//     Term 9 (AT2000-0250)/CC Outputs/Current setpoint value Ch.5 <-> Data Pointer/CurrentSetpointValues[4]
//     Term 9 (AT2000-0250)/CC Outputs/Current setpoint value Ch.6 <-> Data Pointer/CurrentSetpointValues[5]
//     Term 9 (AT2000-0250)/CC Outputs/Current setpoint value Ch.7 <-> Data Pointer/CurrentSetpointValues[6]
//     Term 9 (AT2000-0250)/CC Outputs/Current setpoint value Ch.8 <-> Data Pointer/CurrentSetpointValues[7]
//     Term 9 (AT2000-0250)/CC Outputs/Current setpoint value Ch.9 <-> Data Pointer/CurrentSetpointValues[8]
//     Term 9 (AT2000-0250)/Term 10 (AT2000-5250)/FB Inputs/Value Channel 01 <-> Data Pointer/RawPositionValues[0]
//     Term 9 (AT2000-0250)/Term 10 (AT2000-5250)/FB Inputs/Value Channel 02 <-> Data Pointer/RawPositionValues[1]
//     Term 9 (AT2000-0250)/Term 10 (AT2000-5250)/FB Inputs/Value Channel 03 <-> Data Pointer/RawPositionValues[2]
//     Term 9 (AT2000-0250)/Term 10 (AT2000-5250)/FB Inputs/Value Channel 04 <-> Data Pointer/RawPositionValues[3]
//     Term 9 (AT2000-0250)/Term 10 (AT2000-5250)/FB Inputs/Value Channel 05 <-> Data Pointer/RawPositionValues[4]
//     Term 9 (AT2000-0250)/Term 10 (AT2000-5250)/FB Inputs/Value Channel 06 <-> Data Pointer/RawPositionValues[5]
//     Term 9 (AT2000-0250)/Term 10 (AT2000-5250)/FB Inputs/Value Channel 07 <-> Data Pointer/RawPositionValues[6]
//     Term 9 (AT2000-0250)/Term 10 (AT2000-5250)/FB Inputs/Value Channel 08 <-> Data Pointer/RawPositionValues[7]
//     Term 9 (AT2000-0250)/Term 10 (AT2000-5250)/FB Inputs/Value Channel 09 <-> Data Pointer/RawPositionValues[8]
//     Term 9 (AT2000-0250)/Term 10 (AT2000-5250)/FB Inputs/Value Channel 10 <-> Data Pointer/RawPositionValues[9]
//     Term 9 (AT2000-0250)/Term 10 (AT2000-5250)/FB Inputs/Value Channel 11 <-> Data Pointer/RawPositionValues[10]
//     Term 9 (AT2000-0250)/Term 10 (AT2000-5250)/FB Inputs/Value Channel 12 <-> Data Pointer/RawPositionValues[11]
//     Term 9 (AT2000-0250)/Term 10 (AT2000-5250)/FB Inputs/Value Channel 13 <-> Data Pointer/RawPositionValues[12]
//     Term 9 (AT2000-0250)/Term 10 (AT2000-5250)/FB Inputs/Value Channel 14 <-> Data Pointer/RawPositionValues[13]
//     Term 9 (AT2000-0250)/Term 10 (AT2000-5250)/FB Inputs/Value Channel 15 <-> Data Pointer/RawPositionValues[14]
//     Term 9 (AT2000-0250)/Term 10 (AT2000-5250)/FB Inputs/Value Channel 16 <-> Data Pointer/RawPositionValues[15]
//     Term 9 (AT2000-0250)/Term 10 (AT2000-5250)/FB Inputs/Value Channel 17 <-> Data Pointer/RawPositionValues[16]
//     Term 9 (AT2000-0250)/Term 10 (AT2000-5250)/FB Inputs/Value Channel 18 <-> Data Pointer/RawPositionValues[17]
//     Term 9 (AT2000-0250)/Term 10 (AT2000-5250)/FB Inputs/Value Channel 19 <-> Data Pointer/RawPositionValues[18]
//     Term 9 (AT2000-0250)/Term 10 (AT2000-5250)/FB Inputs/Value Channel 20 <-> Data Pointer/RawPositionValues[19]
//     Term 9 (AT2000-0250)/Term 10 (AT2000-5250)/FB Inputs/Value Channel 21 <-> Data Pointer/RawPositionValues[20]
//     Term 9 (AT2000-0250)/Term 10 (AT2000-5250)/FB Inputs/Value Channel 22 <-> Data Pointer/RawPositionValues[21]
//     Term 9 (AT2000-0250)/Term 10 (AT2000-5250)/FB Inputs/Value Channel 23 <-> Data Pointer/RawPositionValues[22]
//     Term 9 (AT2000-0250)/Term 10 (AT2000-5250)/FB Inputs/Value Channel 24 <-> Data Pointer/RawPositionValues[23]
//     Term 9 (AT2000-0250)/Term 10 (AT2000-5250)/FB Inputs/Value Channel 25 <-> Data Pointer/RawPositionValues[24]
//     Term 9 (AT2000-0250)/Term 10 (AT2000-5250)/FB Inputs/Value Channel 26 <-> Data Pointer/RawPositionValues[25]
//     Term 9 (AT2000-0250)/Term 10 (AT2000-5250)/FB Inputs/Value Channel 27 <-> Data Pointer/RawPositionValues[26]
//     Term 9 (AT2000-0250)/Term 10 (AT2000-5250)/FB Inputs/Value Channel 28 <-> Data Pointer/RawPositionValues[27]
//     Term 9 (AT2000-0250)/Term 10 (AT2000-5250)/FB Inputs/Value Channel 29 <-> Data Pointer/RawPositionValues[28]
//     Term 9 (AT2000-0250)/Term 10 (AT2000-5250)/FB Inputs/Value Channel 30 <-> Data Pointer/RawPositionValues[29]
//     Term 9 (AT2000-0250)/Term 10 (AT2000-5250)/FB Inputs/Value Channel 31 <-> Data Pointer/RawPositionValues[30]
//     Term 9 (AT2000-0250)/Term 10 (AT2000-5250)/FB Inputs/Value Channel 32 <-> Data Pointer/RawPositionValues[31]
//   (this object) <-> TcCOM Objects/XtsProcessingUnit 1/Part 1/Module 6
//     Term 11 (AT2000-0250)/CC Inputs/Current actual value Ch.1 <-> Data Pointer/CurrentActualValues[0]
//     Term 11 (AT2000-0250)/CC Inputs/Current actual value Ch.10 <-> Data Pointer/CurrentActualValues[9]
//     Term 11 (AT2000-0250)/CC Inputs/Current actual value Ch.11 <-> Data Pointer/CurrentActualValues[10]
//     Term 11 (AT2000-0250)/CC Inputs/Current actual value Ch.12 <-> Data Pointer/CurrentActualValues[11]
//     Term 11 (AT2000-0250)/CC Inputs/Current actual value Ch.13 <-> Data Pointer/CurrentActualValues[12]
//     Term 11 (AT2000-0250)/CC Inputs/Current actual value Ch.14 <-> Data Pointer/CurrentActualValues[13]
//     Term 11 (AT2000-0250)/CC Inputs/Current actual value Ch.15 <-> Data Pointer/CurrentActualValues[14]
//     Term 11 (AT2000-0250)/CC Inputs/Current actual value Ch.2 <-> Data Pointer/CurrentActualValues[1]
//     Term 11 (AT2000-0250)/CC Inputs/Current actual value Ch.3 <-> Data Pointer/CurrentActualValues[2]
//     Term 11 (AT2000-0250)/CC Inputs/Current actual value Ch.4 <-> Data Pointer/CurrentActualValues[3]
//     Term 11 (AT2000-0250)/CC Inputs/Current actual value Ch.5 <-> Data Pointer/CurrentActualValues[4]
//     Term 11 (AT2000-0250)/CC Inputs/Current actual value Ch.6 <-> Data Pointer/CurrentActualValues[5]
//     Term 11 (AT2000-0250)/CC Inputs/Current actual value Ch.7 <-> Data Pointer/CurrentActualValues[6]
//     Term 11 (AT2000-0250)/CC Inputs/Current actual value Ch.8 <-> Data Pointer/CurrentActualValues[7]
//     Term 11 (AT2000-0250)/CC Inputs/Current actual value Ch.9 <-> Data Pointer/CurrentActualValues[8]
//     Term 11 (AT2000-0250)/CC Inputs/Status <-> Data Pointer/Status
//     Term 11 (AT2000-0250)/CC Outputs/Control <-> Data Pointer/Control
//     Term 11 (AT2000-0250)/CC Outputs/Current setpoint value Ch.1 <-> Data Pointer/CurrentSetpointValues[0]
//     Term 11 (AT2000-0250)/CC Outputs/Current setpoint value Ch.10 <-> Data Pointer/CurrentSetpointValues[9]
//     Term 11 (AT2000-0250)/CC Outputs/Current setpoint value Ch.11 <-> Data Pointer/CurrentSetpointValues[10]
//     Term 11 (AT2000-0250)/CC Outputs/Current setpoint value Ch.12 <-> Data Pointer/CurrentSetpointValues[11]
//     Term 11 (AT2000-0250)/CC Outputs/Current setpoint value Ch.13 <-> Data Pointer/CurrentSetpointValues[12]
//     Term 11 (AT2000-0250)/CC Outputs/Current setpoint value Ch.14 <-> Data Pointer/CurrentSetpointValues[13]
//     Term 11 (AT2000-0250)/CC Outputs/Current setpoint value Ch.15 <-> Data Pointer/CurrentSetpointValues[14]
//     Term 11 (AT2000-0250)/CC Outputs/Current setpoint value Ch.2 <-> Data Pointer/CurrentSetpointValues[1]
//     Term 11 (AT2000-0250)/CC Outputs/Current setpoint value Ch.3 <-> Data Pointer/CurrentSetpointValues[2]
//     Term 11 (AT2000-0250)/CC Outputs/Current setpoint value Ch.4 <-> Data Pointer/CurrentSetpointValues[3]
//     Term 11 (AT2000-0250)/CC Outputs/Current setpoint value Ch.5 <-> Data Pointer/CurrentSetpointValues[4]
//     Term 11 (AT2000-0250)/CC Outputs/Current setpoint value Ch.6 <-> Data Pointer/CurrentSetpointValues[5]
//     Term 11 (AT2000-0250)/CC Outputs/Current setpoint value Ch.7 <-> Data Pointer/CurrentSetpointValues[6]
//     Term 11 (AT2000-0250)/CC Outputs/Current setpoint value Ch.8 <-> Data Pointer/CurrentSetpointValues[7]
//     Term 11 (AT2000-0250)/CC Outputs/Current setpoint value Ch.9 <-> Data Pointer/CurrentSetpointValues[8]
//     Term 11 (AT2000-0250)/Term 12 (AT2000-5250)/FB Inputs/Value Channel 01 <-> Data Pointer/RawPositionValues[0]
//     Term 11 (AT2000-0250)/Term 12 (AT2000-5250)/FB Inputs/Value Channel 02 <-> Data Pointer/RawPositionValues[1]
//     Term 11 (AT2000-0250)/Term 12 (AT2000-5250)/FB Inputs/Value Channel 03 <-> Data Pointer/RawPositionValues[2]
//     Term 11 (AT2000-0250)/Term 12 (AT2000-5250)/FB Inputs/Value Channel 04 <-> Data Pointer/RawPositionValues[3]
//     Term 11 (AT2000-0250)/Term 12 (AT2000-5250)/FB Inputs/Value Channel 05 <-> Data Pointer/RawPositionValues[4]
//     Term 11 (AT2000-0250)/Term 12 (AT2000-5250)/FB Inputs/Value Channel 06 <-> Data Pointer/RawPositionValues[5]
//     Term 11 (AT2000-0250)/Term 12 (AT2000-5250)/FB Inputs/Value Channel 07 <-> Data Pointer/RawPositionValues[6]
//     Term 11 (AT2000-0250)/Term 12 (AT2000-5250)/FB Inputs/Value Channel 08 <-> Data Pointer/RawPositionValues[7]
//     Term 11 (AT2000-0250)/Term 12 (AT2000-5250)/FB Inputs/Value Channel 09 <-> Data Pointer/RawPositionValues[8]
//     Term 11 (AT2000-0250)/Term 12 (AT2000-5250)/FB Inputs/Value Channel 10 <-> Data Pointer/RawPositionValues[9]
//     Term 11 (AT2000-0250)/Term 12 (AT2000-5250)/FB Inputs/Value Channel 11 <-> Data Pointer/RawPositionValues[10]
//     Term 11 (AT2000-0250)/Term 12 (AT2000-5250)/FB Inputs/Value Channel 12 <-> Data Pointer/RawPositionValues[11]
//     Term 11 (AT2000-0250)/Term 12 (AT2000-5250)/FB Inputs/Value Channel 13 <-> Data Pointer/RawPositionValues[12]
//     Term 11 (AT2000-0250)/Term 12 (AT2000-5250)/FB Inputs/Value Channel 14 <-> Data Pointer/RawPositionValues[13]
//     Term 11 (AT2000-0250)/Term 12 (AT2000-5250)/FB Inputs/Value Channel 15 <-> Data Pointer/RawPositionValues[14]
//     Term 11 (AT2000-0250)/Term 12 (AT2000-5250)/FB Inputs/Value Channel 16 <-> Data Pointer/RawPositionValues[15]
//     Term 11 (AT2000-0250)/Term 12 (AT2000-5250)/FB Inputs/Value Channel 17 <-> Data Pointer/RawPositionValues[16]
//     Term 11 (AT2000-0250)/Term 12 (AT2000-5250)/FB Inputs/Value Channel 18 <-> Data Pointer/RawPositionValues[17]
//     Term 11 (AT2000-0250)/Term 12 (AT2000-5250)/FB Inputs/Value Channel 19 <-> Data Pointer/RawPositionValues[18]
//     Term 11 (AT2000-0250)/Term 12 (AT2000-5250)/FB Inputs/Value Channel 20 <-> Data Pointer/RawPositionValues[19]
//     Term 11 (AT2000-0250)/Term 12 (AT2000-5250)/FB Inputs/Value Channel 21 <-> Data Pointer/RawPositionValues[20]
//     Term 11 (AT2000-0250)/Term 12 (AT2000-5250)/FB Inputs/Value Channel 22 <-> Data Pointer/RawPositionValues[21]
//     Term 11 (AT2000-0250)/Term 12 (AT2000-5250)/FB Inputs/Value Channel 23 <-> Data Pointer/RawPositionValues[22]
//     Term 11 (AT2000-0250)/Term 12 (AT2000-5250)/FB Inputs/Value Channel 24 <-> Data Pointer/RawPositionValues[23]
//     Term 11 (AT2000-0250)/Term 12 (AT2000-5250)/FB Inputs/Value Channel 25 <-> Data Pointer/RawPositionValues[24]
//     Term 11 (AT2000-0250)/Term 12 (AT2000-5250)/FB Inputs/Value Channel 26 <-> Data Pointer/RawPositionValues[25]
//     Term 11 (AT2000-0250)/Term 12 (AT2000-5250)/FB Inputs/Value Channel 27 <-> Data Pointer/RawPositionValues[26]
//     Term 11 (AT2000-0250)/Term 12 (AT2000-5250)/FB Inputs/Value Channel 28 <-> Data Pointer/RawPositionValues[27]
//     Term 11 (AT2000-0250)/Term 12 (AT2000-5250)/FB Inputs/Value Channel 29 <-> Data Pointer/RawPositionValues[28]
//     Term 11 (AT2000-0250)/Term 12 (AT2000-5250)/FB Inputs/Value Channel 30 <-> Data Pointer/RawPositionValues[29]
//     Term 11 (AT2000-0250)/Term 12 (AT2000-5250)/FB Inputs/Value Channel 31 <-> Data Pointer/RawPositionValues[30]
//     Term 11 (AT2000-0250)/Term 12 (AT2000-5250)/FB Inputs/Value Channel 32 <-> Data Pointer/RawPositionValues[31]
//   (this object) <-> TcCOM Objects/XtsProcessingUnit 1/Part 1/Module 7
//     Term 13 (AT2050-0500)/CC Inputs/Current actual value Ch.1 <-> Data Pointer/CurrentActualValues[0]
//     Term 13 (AT2050-0500)/CC Inputs/Current actual value Ch.10 <-> Data Pointer/CurrentActualValues[9]
//     Term 13 (AT2050-0500)/CC Inputs/Current actual value Ch.11 <-> Data Pointer/CurrentActualValues[10]
//     Term 13 (AT2050-0500)/CC Inputs/Current actual value Ch.12 <-> Data Pointer/CurrentActualValues[11]
//     Term 13 (AT2050-0500)/CC Inputs/Current actual value Ch.13 <-> Data Pointer/CurrentActualValues[12]
//     Term 13 (AT2050-0500)/CC Inputs/Current actual value Ch.14 <-> Data Pointer/CurrentActualValues[13]
//     Term 13 (AT2050-0500)/CC Inputs/Current actual value Ch.15 <-> Data Pointer/CurrentActualValues[14]
//     Term 13 (AT2050-0500)/CC Inputs/Current actual value Ch.2 <-> Data Pointer/CurrentActualValues[1]
//     Term 13 (AT2050-0500)/CC Inputs/Current actual value Ch.3 <-> Data Pointer/CurrentActualValues[2]
//     Term 13 (AT2050-0500)/CC Inputs/Current actual value Ch.4 <-> Data Pointer/CurrentActualValues[3]
//     Term 13 (AT2050-0500)/CC Inputs/Current actual value Ch.5 <-> Data Pointer/CurrentActualValues[4]
//     Term 13 (AT2050-0500)/CC Inputs/Current actual value Ch.6 <-> Data Pointer/CurrentActualValues[5]
//     Term 13 (AT2050-0500)/CC Inputs/Current actual value Ch.7 <-> Data Pointer/CurrentActualValues[6]
//     Term 13 (AT2050-0500)/CC Inputs/Current actual value Ch.8 <-> Data Pointer/CurrentActualValues[7]
//     Term 13 (AT2050-0500)/CC Inputs/Current actual value Ch.9 <-> Data Pointer/CurrentActualValues[8]
//     Term 13 (AT2050-0500)/CC Inputs/Status <-> Data Pointer/Status
//     Term 13 (AT2050-0500)/CC Outputs/Control <-> Data Pointer/Control
//     Term 13 (AT2050-0500)/CC Outputs/Current setpoint value Ch.1 <-> Data Pointer/CurrentSetpointValues[0]
//     Term 13 (AT2050-0500)/CC Outputs/Current setpoint value Ch.10 <-> Data Pointer/CurrentSetpointValues[9]
//     Term 13 (AT2050-0500)/CC Outputs/Current setpoint value Ch.11 <-> Data Pointer/CurrentSetpointValues[10]
//     Term 13 (AT2050-0500)/CC Outputs/Current setpoint value Ch.12 <-> Data Pointer/CurrentSetpointValues[11]
//     Term 13 (AT2050-0500)/CC Outputs/Current setpoint value Ch.13 <-> Data Pointer/CurrentSetpointValues[12]
//     Term 13 (AT2050-0500)/CC Outputs/Current setpoint value Ch.14 <-> Data Pointer/CurrentSetpointValues[13]
//     Term 13 (AT2050-0500)/CC Outputs/Current setpoint value Ch.15 <-> Data Pointer/CurrentSetpointValues[14]
//     Term 13 (AT2050-0500)/CC Outputs/Current setpoint value Ch.2 <-> Data Pointer/CurrentSetpointValues[1]
//     Term 13 (AT2050-0500)/CC Outputs/Current setpoint value Ch.3 <-> Data Pointer/CurrentSetpointValues[2]
//     Term 13 (AT2050-0500)/CC Outputs/Current setpoint value Ch.4 <-> Data Pointer/CurrentSetpointValues[3]
//     Term 13 (AT2050-0500)/CC Outputs/Current setpoint value Ch.5 <-> Data Pointer/CurrentSetpointValues[4]
//     Term 13 (AT2050-0500)/CC Outputs/Current setpoint value Ch.6 <-> Data Pointer/CurrentSetpointValues[5]
//     Term 13 (AT2050-0500)/CC Outputs/Current setpoint value Ch.7 <-> Data Pointer/CurrentSetpointValues[6]
//     Term 13 (AT2050-0500)/CC Outputs/Current setpoint value Ch.8 <-> Data Pointer/CurrentSetpointValues[7]
//     Term 13 (AT2050-0500)/CC Outputs/Current setpoint value Ch.9 <-> Data Pointer/CurrentSetpointValues[8]
//     Term 13 (AT2050-0500)/Term 14 (AT2050-5500)/FB Inputs/Value Channel 01 <-> Data Pointer/RawPositionValues[0]
//     Term 13 (AT2050-0500)/Term 14 (AT2050-5500)/FB Inputs/Value Channel 02 <-> Data Pointer/RawPositionValues[1]
//     Term 13 (AT2050-0500)/Term 14 (AT2050-5500)/FB Inputs/Value Channel 03 <-> Data Pointer/RawPositionValues[2]
//     Term 13 (AT2050-0500)/Term 14 (AT2050-5500)/FB Inputs/Value Channel 04 <-> Data Pointer/RawPositionValues[3]
//     Term 13 (AT2050-0500)/Term 14 (AT2050-5500)/FB Inputs/Value Channel 05 <-> Data Pointer/RawPositionValues[4]
//     Term 13 (AT2050-0500)/Term 14 (AT2050-5500)/FB Inputs/Value Channel 06 <-> Data Pointer/RawPositionValues[5]
//     Term 13 (AT2050-0500)/Term 14 (AT2050-5500)/FB Inputs/Value Channel 07 <-> Data Pointer/RawPositionValues[6]
//     Term 13 (AT2050-0500)/Term 14 (AT2050-5500)/FB Inputs/Value Channel 08 <-> Data Pointer/RawPositionValues[7]
//     Term 13 (AT2050-0500)/Term 14 (AT2050-5500)/FB Inputs/Value Channel 09 <-> Data Pointer/RawPositionValues[8]
//     Term 13 (AT2050-0500)/Term 14 (AT2050-5500)/FB Inputs/Value Channel 10 <-> Data Pointer/RawPositionValues[9]
//     Term 13 (AT2050-0500)/Term 14 (AT2050-5500)/FB Inputs/Value Channel 11 <-> Data Pointer/RawPositionValues[10]
//     Term 13 (AT2050-0500)/Term 14 (AT2050-5500)/FB Inputs/Value Channel 12 <-> Data Pointer/RawPositionValues[11]
//     Term 13 (AT2050-0500)/Term 14 (AT2050-5500)/FB Inputs/Value Channel 13 <-> Data Pointer/RawPositionValues[12]
//     Term 13 (AT2050-0500)/Term 14 (AT2050-5500)/FB Inputs/Value Channel 14 <-> Data Pointer/RawPositionValues[13]
//     Term 13 (AT2050-0500)/Term 14 (AT2050-5500)/FB Inputs/Value Channel 15 <-> Data Pointer/RawPositionValues[14]
//     Term 13 (AT2050-0500)/Term 14 (AT2050-5500)/FB Inputs/Value Channel 16 <-> Data Pointer/RawPositionValues[15]
//     Term 13 (AT2050-0500)/Term 14 (AT2050-5500)/FB Inputs/Value Channel 17 <-> Data Pointer/RawPositionValues[16]
//     Term 13 (AT2050-0500)/Term 14 (AT2050-5500)/FB Inputs/Value Channel 18 <-> Data Pointer/RawPositionValues[17]
//     Term 13 (AT2050-0500)/Term 14 (AT2050-5500)/FB Inputs/Value Channel 19 <-> Data Pointer/RawPositionValues[18]
//     Term 13 (AT2050-0500)/Term 14 (AT2050-5500)/FB Inputs/Value Channel 20 <-> Data Pointer/RawPositionValues[19]
//     Term 13 (AT2050-0500)/Term 14 (AT2050-5500)/FB Inputs/Value Channel 21 <-> Data Pointer/RawPositionValues[20]
//     Term 13 (AT2050-0500)/Term 14 (AT2050-5500)/FB Inputs/Value Channel 22 <-> Data Pointer/RawPositionValues[21]
//     Term 13 (AT2050-0500)/Term 14 (AT2050-5500)/FB Inputs/Value Channel 23 <-> Data Pointer/RawPositionValues[22]
//     Term 13 (AT2050-0500)/Term 14 (AT2050-5500)/FB Inputs/Value Channel 24 <-> Data Pointer/RawPositionValues[23]
//     Term 13 (AT2050-0500)/Term 14 (AT2050-5500)/FB Inputs/Value Channel 25 <-> Data Pointer/RawPositionValues[24]
//     Term 13 (AT2050-0500)/Term 14 (AT2050-5500)/FB Inputs/Value Channel 26 <-> Data Pointer/RawPositionValues[25]
//     Term 13 (AT2050-0500)/Term 14 (AT2050-5500)/FB Inputs/Value Channel 27 <-> Data Pointer/RawPositionValues[26]
//     Term 13 (AT2050-0500)/Term 14 (AT2050-5500)/FB Inputs/Value Channel 28 <-> Data Pointer/RawPositionValues[27]
//     Term 13 (AT2050-0500)/Term 14 (AT2050-5500)/FB Inputs/Value Channel 29 <-> Data Pointer/RawPositionValues[28]
//     Term 13 (AT2050-0500)/Term 14 (AT2050-5500)/FB Inputs/Value Channel 30 <-> Data Pointer/RawPositionValues[29]
//     Term 13 (AT2050-0500)/Term 14 (AT2050-5500)/FB Inputs/Value Channel 31 <-> Data Pointer/RawPositionValues[30]
//     Term 13 (AT2050-0500)/Term 14 (AT2050-5500)/FB Inputs/Value Channel 32 <-> Data Pointer/RawPositionValues[31]
//   (this object) <-> TcCOM Objects/XtsProcessingUnit 1/Part 1/Module 8
//     Term 15 (AT2050-0501)/CC Inputs/Current actual value Ch.1 <-> Data Pointer/CurrentActualValues[0]
//     Term 15 (AT2050-0501)/CC Inputs/Current actual value Ch.10 <-> Data Pointer/CurrentActualValues[9]
//     Term 15 (AT2050-0501)/CC Inputs/Current actual value Ch.11 <-> Data Pointer/CurrentActualValues[10]
//     Term 15 (AT2050-0501)/CC Inputs/Current actual value Ch.12 <-> Data Pointer/CurrentActualValues[11]
//     Term 15 (AT2050-0501)/CC Inputs/Current actual value Ch.13 <-> Data Pointer/CurrentActualValues[12]
//     Term 15 (AT2050-0501)/CC Inputs/Current actual value Ch.14 <-> Data Pointer/CurrentActualValues[13]
//     Term 15 (AT2050-0501)/CC Inputs/Current actual value Ch.15 <-> Data Pointer/CurrentActualValues[14]
//     Term 15 (AT2050-0501)/CC Inputs/Current actual value Ch.2 <-> Data Pointer/CurrentActualValues[1]
//     Term 15 (AT2050-0501)/CC Inputs/Current actual value Ch.3 <-> Data Pointer/CurrentActualValues[2]
//     Term 15 (AT2050-0501)/CC Inputs/Current actual value Ch.4 <-> Data Pointer/CurrentActualValues[3]
//     Term 15 (AT2050-0501)/CC Inputs/Current actual value Ch.5 <-> Data Pointer/CurrentActualValues[4]
//     Term 15 (AT2050-0501)/CC Inputs/Current actual value Ch.6 <-> Data Pointer/CurrentActualValues[5]
//     Term 15 (AT2050-0501)/CC Inputs/Current actual value Ch.7 <-> Data Pointer/CurrentActualValues[6]
//     Term 15 (AT2050-0501)/CC Inputs/Current actual value Ch.8 <-> Data Pointer/CurrentActualValues[7]
//     Term 15 (AT2050-0501)/CC Inputs/Current actual value Ch.9 <-> Data Pointer/CurrentActualValues[8]
//     Term 15 (AT2050-0501)/CC Inputs/Status <-> Data Pointer/Status
//     Term 15 (AT2050-0501)/CC Outputs/Control <-> Data Pointer/Control
//     Term 15 (AT2050-0501)/CC Outputs/Current setpoint value Ch.1 <-> Data Pointer/CurrentSetpointValues[0]
//     Term 15 (AT2050-0501)/CC Outputs/Current setpoint value Ch.10 <-> Data Pointer/CurrentSetpointValues[9]
//     Term 15 (AT2050-0501)/CC Outputs/Current setpoint value Ch.11 <-> Data Pointer/CurrentSetpointValues[10]
//     Term 15 (AT2050-0501)/CC Outputs/Current setpoint value Ch.12 <-> Data Pointer/CurrentSetpointValues[11]
//     Term 15 (AT2050-0501)/CC Outputs/Current setpoint value Ch.13 <-> Data Pointer/CurrentSetpointValues[12]
//     Term 15 (AT2050-0501)/CC Outputs/Current setpoint value Ch.14 <-> Data Pointer/CurrentSetpointValues[13]
//     Term 15 (AT2050-0501)/CC Outputs/Current setpoint value Ch.15 <-> Data Pointer/CurrentSetpointValues[14]
//     Term 15 (AT2050-0501)/CC Outputs/Current setpoint value Ch.2 <-> Data Pointer/CurrentSetpointValues[1]
//     Term 15 (AT2050-0501)/CC Outputs/Current setpoint value Ch.3 <-> Data Pointer/CurrentSetpointValues[2]
//     Term 15 (AT2050-0501)/CC Outputs/Current setpoint value Ch.4 <-> Data Pointer/CurrentSetpointValues[3]
//     Term 15 (AT2050-0501)/CC Outputs/Current setpoint value Ch.5 <-> Data Pointer/CurrentSetpointValues[4]
//     Term 15 (AT2050-0501)/CC Outputs/Current setpoint value Ch.6 <-> Data Pointer/CurrentSetpointValues[5]
//     Term 15 (AT2050-0501)/CC Outputs/Current setpoint value Ch.7 <-> Data Pointer/CurrentSetpointValues[6]
//     Term 15 (AT2050-0501)/CC Outputs/Current setpoint value Ch.8 <-> Data Pointer/CurrentSetpointValues[7]
//     Term 15 (AT2050-0501)/CC Outputs/Current setpoint value Ch.9 <-> Data Pointer/CurrentSetpointValues[8]
//     Term 15 (AT2050-0501)/Term 16 (AT2050-5501)/FB Inputs/Value Channel 01 <-> Data Pointer/RawPositionValues[0]
//     Term 15 (AT2050-0501)/Term 16 (AT2050-5501)/FB Inputs/Value Channel 02 <-> Data Pointer/RawPositionValues[1]
//     Term 15 (AT2050-0501)/Term 16 (AT2050-5501)/FB Inputs/Value Channel 03 <-> Data Pointer/RawPositionValues[2]
//     Term 15 (AT2050-0501)/Term 16 (AT2050-5501)/FB Inputs/Value Channel 04 <-> Data Pointer/RawPositionValues[3]
//     Term 15 (AT2050-0501)/Term 16 (AT2050-5501)/FB Inputs/Value Channel 05 <-> Data Pointer/RawPositionValues[4]
//     Term 15 (AT2050-0501)/Term 16 (AT2050-5501)/FB Inputs/Value Channel 06 <-> Data Pointer/RawPositionValues[5]
//     Term 15 (AT2050-0501)/Term 16 (AT2050-5501)/FB Inputs/Value Channel 07 <-> Data Pointer/RawPositionValues[6]
//     Term 15 (AT2050-0501)/Term 16 (AT2050-5501)/FB Inputs/Value Channel 08 <-> Data Pointer/RawPositionValues[7]
//     Term 15 (AT2050-0501)/Term 16 (AT2050-5501)/FB Inputs/Value Channel 09 <-> Data Pointer/RawPositionValues[8]
//     Term 15 (AT2050-0501)/Term 16 (AT2050-5501)/FB Inputs/Value Channel 10 <-> Data Pointer/RawPositionValues[9]
//     Term 15 (AT2050-0501)/Term 16 (AT2050-5501)/FB Inputs/Value Channel 11 <-> Data Pointer/RawPositionValues[10]
//     Term 15 (AT2050-0501)/Term 16 (AT2050-5501)/FB Inputs/Value Channel 12 <-> Data Pointer/RawPositionValues[11]
//     Term 15 (AT2050-0501)/Term 16 (AT2050-5501)/FB Inputs/Value Channel 13 <-> Data Pointer/RawPositionValues[12]
//     Term 15 (AT2050-0501)/Term 16 (AT2050-5501)/FB Inputs/Value Channel 14 <-> Data Pointer/RawPositionValues[13]
//     Term 15 (AT2050-0501)/Term 16 (AT2050-5501)/FB Inputs/Value Channel 15 <-> Data Pointer/RawPositionValues[14]
//     Term 15 (AT2050-0501)/Term 16 (AT2050-5501)/FB Inputs/Value Channel 16 <-> Data Pointer/RawPositionValues[15]
//     Term 15 (AT2050-0501)/Term 16 (AT2050-5501)/FB Inputs/Value Channel 17 <-> Data Pointer/RawPositionValues[16]
//     Term 15 (AT2050-0501)/Term 16 (AT2050-5501)/FB Inputs/Value Channel 18 <-> Data Pointer/RawPositionValues[17]
//     Term 15 (AT2050-0501)/Term 16 (AT2050-5501)/FB Inputs/Value Channel 19 <-> Data Pointer/RawPositionValues[18]
//     Term 15 (AT2050-0501)/Term 16 (AT2050-5501)/FB Inputs/Value Channel 20 <-> Data Pointer/RawPositionValues[19]
//     Term 15 (AT2050-0501)/Term 16 (AT2050-5501)/FB Inputs/Value Channel 21 <-> Data Pointer/RawPositionValues[20]
//     Term 15 (AT2050-0501)/Term 16 (AT2050-5501)/FB Inputs/Value Channel 22 <-> Data Pointer/RawPositionValues[21]
//     Term 15 (AT2050-0501)/Term 16 (AT2050-5501)/FB Inputs/Value Channel 23 <-> Data Pointer/RawPositionValues[22]
//     Term 15 (AT2050-0501)/Term 16 (AT2050-5501)/FB Inputs/Value Channel 24 <-> Data Pointer/RawPositionValues[23]
//     Term 15 (AT2050-0501)/Term 16 (AT2050-5501)/FB Inputs/Value Channel 25 <-> Data Pointer/RawPositionValues[24]
//     Term 15 (AT2050-0501)/Term 16 (AT2050-5501)/FB Inputs/Value Channel 26 <-> Data Pointer/RawPositionValues[25]
//     Term 15 (AT2050-0501)/Term 16 (AT2050-5501)/FB Inputs/Value Channel 27 <-> Data Pointer/RawPositionValues[26]
//     Term 15 (AT2050-0501)/Term 16 (AT2050-5501)/FB Inputs/Value Channel 28 <-> Data Pointer/RawPositionValues[27]
//     Term 15 (AT2050-0501)/Term 16 (AT2050-5501)/FB Inputs/Value Channel 29 <-> Data Pointer/RawPositionValues[28]
//     Term 15 (AT2050-0501)/Term 16 (AT2050-5501)/FB Inputs/Value Channel 30 <-> Data Pointer/RawPositionValues[29]
//     Term 15 (AT2050-0501)/Term 16 (AT2050-5501)/FB Inputs/Value Channel 31 <-> Data Pointer/RawPositionValues[30]
//     Term 15 (AT2050-0501)/Term 16 (AT2050-5501)/FB Inputs/Value Channel 32 <-> Data Pointer/RawPositionValues[31]

CONFIGURATION Main
    RESOURCE PLC ON TwinCAT3
        TASK PlcTask(INTERVAL := T#1ms, PRIORITY := 6);
        PROGRAM MAIN WITH PlcTask : MAIN;
    END_RESOURCE
END_CONFIGURATION

// ---- DUTs/MachineCmd_typ.TcDUT
TYPE MachineCmd_typ :
STRUCT
	Enable		: BOOL;
	Start		: BOOL;
	Stop		: BOOL;
END_STRUCT
END_TYPE

// ---- DUTs/MachineState_enum.TcDUT
{attribute 'strict'}
{attribute 'to_string'}
TYPE MachineState_enum :
(
	MS_OFF		 		:= 0,
	MS_RESTARTING		:= 1,
	MS_ENABLED			:= 2,
	MS_ONESHOT_RECOVER	:= 3,
	MS_RECOVERING		:= 4,
	MS_RUNNING			:= 5,
	MS_CYCLESTOP		:= 6,
	MS_STOPPING			:= 7,
	MS_ERROR			:= 8
);
END_TYPE

// ---- GVLs/GVL.TcGVL
{attribute 'qualified_only'}
VAR_GLOBAL
	newCallTime: LREAL;
END_VAR

// ---- GVLs/Param.TcGVL
{attribute 'qualified_only'}
VAR_GLOBAL CONSTANT
	TRACK_LENGTH 			: LREAL := 4000; // This should be set to the exact length [mm] of the track system
		
	MAX_MOVERS   			: USINT := 100;   // This is the maximum number of movers that can be added to the system
	
	// The following should be set to a value **equal to or greater than** the number of objectives needed
	NUM_MOVERLISTS			: USINT := 10;	// Mover Lists
	NUM_POSITIONTRIGGERS	: USINT := 10;	// Position Triggers
	NUM_STATIONS			: USINT := 10;	// Stations
	NUM_ZONES				: USINT := 10;	// Zones
	
	NUM_TRACKS				: USINT	:= 1;	// Tracks (Typically 1)

	PART_ARRAY_SIZE			: UDINT := 100;
	AUTO_POPULATE_STATIONS  : BOOL := TRUE; // use the Station[x] array to label stations on the visualization. Turn off if manually entering stations in the configurator.
	
	// statistics weighted average
	ALPHA_EMA				: LREAL := 0.1;
END_VAR

// ---- POUs/MAIN.TcPOU
PROGRAM MAIN
VAR	
	// declare XTS with <number of movers>
	XTS				: FB_XTS<6>;
	MainCommands	: MachineCmd_typ;
	// Machine
	State			: MachineState_enum;

	Init			: BOOL;
	// ========= Example Application Variables =========

    nextStation 			: USINT := 4;
                    	
    lowVelocity    			: LREAL := 200;  	// mm/s
    mediumVelocity 			: LREAL := 800;  	// mm/s
    highVelocity   			: LREAL := 1200; 	// mm/s
	
	StationTimer 			: ARRAY[0..Param.NUM_STATIONS] OF TON; // timer blocks, for station dwells
	InitialParameterSet		: MotionParameters_typ;
	RecoveryComplete		: BOOL;
	
	mcDirectionPositive		: Tc2_MC2.MC_Direction;
	Trig0MoverIndex			: UDINT;
	Trig0MoverPosLag		: LREAL;
END_VAR


(* ======================================================================================

--- XTS Starter Project ---

This MAIN (PRG) is intended to serve as an example, which can be modified to suit your specific application.

No programming changes should be necessary inside the provided XTS objects / function block definitions.
They are intended to be simply instantiated and controlled via the provided methods and properties.
However the objects are provided as open-source for modification and extension as needed.

Documentation for these objects can be found online at:
https://beckhoff-usa-community.github.io/XTS_Base/

Bug reports, new feature requests, and general feedback is always welcome on our Github page.
For any other questions, please reach out to your local Application Engineer.

- XTS Application Group | Beckhoff USA

====================================================================================== *)

(*
All sample code provided by Beckhoff Automation LLC are for illustrative purposes only
and are provided “as is” and without any warranties, express or implied. Actual
implementations in applications will vary significantly. Beckhoff Automation LLC shall
have no liability for, and does not waive any rights in relation to, any code samples that it
provides or the use of such code samples for any purpose.
*)



IF NOT Init THEN Initializing(); END_IF

CASE State OF 

	MS_OFF:
		IF MainCommands.Enable THEN
			XTS.Enable				:= TRUE;
			State					:= MS_RESTARTING;
		END_IF

	MS_RESTARTING:
		IF NOT MainCommands.Enable THEN
			XTS.Enable				:= FALSE;
			State					:= MS_STOPPING;
		ELSIF XTS.State = XTS_ENABLED THEN
			State		:= MS_ENABLED;
		END_IF
	
	MS_ENABLED:
		IF NOT MainCommands.Enable THEN
			XTS.Enable				:= FALSE;
			State					:= MS_STOPPING;
		ELSIF MainCommands.Start THEN
			State					:= MS_ONESHOT_RECOVER;
		END_IF
		
	MS_ONESHOT_RECOVER:
		// one time commands before starting typical process motions
		RecoverOneshot();
		State := MS_RECOVERING;
		
	MS_RECOVERING:
		// wait for any recovery actions to complete
		Recovering();
		// test for errors, commands or recovery complete
		IF MainCommands.Stop THEN
			MainCommands.Start		:= FALSE;
			XTS.System.CompleteMoverList.HaltAll();
            State         	:= MS_STOPPING;
        ELSIF NOT MainCommands.Enable THEN
            XTS.Enable		:= FALSE;
			XTS.System.CompleteMoverList.HaltAll();
            State          			:= MS_STOPPING;
		ELSIF RecoveryComplete THEN
			// recovery sequence is complete, move on to run state
			State					:= MS_RUNNING;
        END_IF

	MS_RUNNING:
		// run the station-to-station mover logic
		StationLogic();
		
		// monitor for disable
		IF NOT MainCommands.Enable THEN
			XTS.Enable				:= FALSE;
			XTS.System.CompleteMoverList.HaltAll();
			State					:= MS_STOPPING;
		ELSIF MainCommands.Stop THEN
			MainCommands.Start		:= FALSE;
			XTS.System.CompleteMoverList.HaltAll();
			State					:= MS_STOPPING;
		END_IF

	MS_STOPPING:
		IF NOT MainCommands.Enable THEN
			XTS.Enable 				:= FALSE;
		END_IF
		IF XTS.State = XTS_DISABLED THEN
			State					:= MS_OFF;
		ELSIF  MainCommands.Start THEN
			MainCommands.Stop		:= FALSE;
			State					:= MS_ONESHOT_RECOVER;
		END_IF
	
END_CASE

XTS.CyclicLogic();

ACTION Initializing:
// XTS Object Init
XTS.Station[0].Position 		:= 5;
XTS.Station[1].Position 		:= 750;
XTS.Station[2].Position 		:= 1200;
XTS.Station[3].Position 		:= 1300;
XTS.Station[4].Position 		:= 1400;

XTS.PositionTrigger[0].Position := 1500;
XTS.PositionTrigger[1].Position := 2000;
XTS.PositionTrigger[2].Position := 3500;

XTS.Zone[0].StartPosition		:= 3750;
XTS.Zone[0].EndPosition   		:= 750;

XTS.Zone[1].StartPosition 		:= 750;
XTS.Zone[1].EndPosition   		:= 1750;

XTS.Zone[2].StartPosition 		:= 1750;
XTS.Zone[2].EndPosition   		:= 2750;

XTS.Zone[3].StartPosition		:= 2750;
XTS.Zone[3].EndPosition   		:= 3750;

XTS.InitialParameterSet.Velocity		:= 1000;		// mm/s
XTS.InitialParameterSet.Acceleration	:= 10_000;		// mm/s2
XTS.InitialParameterSet.Deceleration	:= 10_000;		// mm/s2
XTS.InitialParameterSet.Jerk			:= 100_000;		// mm/s3
XTS.InitialParameterSet.Gap				:= 85;			// mm
XTS.InitialParameterSet.Direction		:= Tc3_Mc3Definitions.MC_Direction.mcDirectionPositive;

LowVelocity		:= 300;
MediumVelocity	:= 800;
HighVelocity	:= 1200;

Init	:= TRUE;
END_ACTION

ACTION Recovering:
// this state is called until all movers have completed their desired recovery tasks

// wait for all movers to reach the standstill state and one mover at station 0
IF (XTS.System.CompleteMoverList.IsAllMoversHalted AND XTS.Station[0].MoverInPosition) THEN
	RecoveryComplete := TRUE;
END_IF
END_ACTION

ACTION RecoverOneshot:
// this action is called one time after the start command is issued
// it is intended to provide a single command to each mover to facilitate recovery
// other commands such as resetting counters and timers should also be carried out here

// send all movers to station 0
XTS.System.CompleteMoverList.SetAllVelocity(mediumVelocity).MoveAllToStation( XTS.Station[0] );
XTS.System.ResetStatistics();

// Reinit nextStation
nextStation := 4;
END_ACTION

ACTION StationLogic:
		(*Mover routing logic should be written here to define the system's operating behavior.
		Station implementations, Position Trigger logic, etc. In general, you can remove the example code
		here down to the short line break that looks like this: // ============= *)
	
        // Station 0 Logic
        IF XTS.Station[0].MoverInPosition THEN
            StationTimer[0](IN := TRUE, PT := T#1000MS);
            IF StationTimer[0].Q THEN
                XTS.Mover[XTS.Station[0].CurrentMover.MoverIndex].MoveToStationByRampTime(
					DestinationStation:= XTS.Station[1], 
					Velocity:= 500, 
					RampTime:= 1.5, 
					Stiffness:= 0.5, 
					Gap:= 85);
            END_IF
        ELSE
            StationTimer[0](IN := FALSE);
        END_IF
		
        // Station 1 Logic		
        IF XTS.Station[1].MoverInPosition THEN
            StationTimer[1](IN := TRUE, PT := T#250MS);
            IF StationTimer[1].Q THEN
                XTS.Station[1].CurrentMover.MoveToStation(XTS.Station[nextStation]);
                nextStation := nextStation - 1;
                IF nextStation = 1 THEN
                    nextStation := 4;
                END_IF
            END_IF
        ELSE
            StationTimer[1](IN := FALSE);
        END_IF
		
		// Group of Stations 2, 3, and 4 Logic
        IF XTS.Station[2].MoverInPosition AND XTS.Station[3].MoverInPosition AND XTS.Station[4].MoverInPosition THEN
            StationTimer[2](IN := TRUE, PT := T#750MS);
            IF StationTimer[2].Q THEN
				StationTimer[2](IN := FALSE);
				
				XTS.Station[2].CurrentMover.MotionParameters:= XTS.InitialParameterSet;
				XTS.Station[3].CurrentMover.MotionParameters:= XTS.InitialParameterSet;
				XTS.Station[4].CurrentMover.MotionParameters:= XTS.InitialParameterSet;

                XTS.Station[2].CurrentMover.MoveVelocity(500);
                XTS.Station[3].CurrentMover.MoveVelocity(500);
                XTS.Station[4].CurrentMover.MoveVelocity(500);
				
            END_IF
        END_IF
		
        // Position Trigger 0 Logic
        IF XTS.PositionTrigger[0].MoverPassedPosition THEN
            XTS.PositionTrigger[0].CurrentMover.SetVelocity(lowVelocity);
			
			// To Call ApplicationMover addon Method/Properties/Variables, you must call Mover[] array index directly
			// Get MoverIndex for later use with ApplicationMover addons
			Trig0MoverIndex		:= XTS.PositionTrigger[0].CurrentMover.MoverIndex;
			
			// Call ApplicationMover Method/Properties/Variables using previously latched MoverIndex
			Trig0MoverPosLag	:= XTS.Mover[Trig0MoverIndex].PositionLag;
			
            XTS.PositionTrigger[0].MuteCurrent();
						
        END_IF
		
        // Position Trigger 1 Logic
        IF XTS.PositionTrigger[1].MoverPassedPosition THEN
			XTS.PositionTrigger[1].CurrentMover.SetAcceleration(5E2);
            XTS.PositionTrigger[1].CurrentMover.SetVelocity(highVelocity);
            XTS.PositionTrigger[1].MuteCurrent();
        END_IF

		// Position Trigger 2 Logic
        IF XTS.PositionTrigger[2].MoverPassedPosition THEN
			XTS.PositionTrigger[2].CurrentMover.SetAcceleration(1E4);
            XTS.PositionTrigger[2].CurrentMover.SetVelocity(lowVelocity);
            XTS.PositionTrigger[2].CurrentMover.MoveToStation(XTS.Station[0]);
            XTS.PositionTrigger[2].MuteCurrent();
        END_IF
END_ACTION

END_PROGRAM

// ---- POUs/ApplicationMover.TcPOU
// This function Block extends the Referenced Library Mover (FB), so the user can expand the capabilities of the XTS Mover Functions
FUNCTION_BLOCK ApplicationMover EXTENDS Mover
VAR_INPUT
END_VAR
VAR_OUTPUT
END_VAR
VAR
	cnt: UDINT;
	_PositionLag: LREAL;
	fbMC_CalcDynamicsByRampTime: MC_CalcDynamicsByRampTime;
END_VAR

METHOD Cyclic : iMover
VAR_IN_OUT
	GroupReference	: AXES_GROUP_REF;
END_VAR
// Call Base Class (Mover) Cyclic Logic
SUPER^.Cyclic(GroupReference);

//======= 
// To Call ApplicationMover addon Method/Properties/Variables... 
//		you must call Mover[] array index directly, as Station/Zone/PositionTrig/SpeedTrig do not know about ApplicationMover add ons

// Add ApplicationMover specific code here
cnt:= cnt + 1;
_PositionLag:= THIS^.AxisReference.NcToPlc.PosDiff;



// Latch Errors
IF fbMC_CalcDynamicsByRampTime.Error THEN
	ErrorID						:= fbMC_CalcDynamicsByRampTime.ErrorID;
	ErrorOrigin					:= CONCAT( InstancePath, '.fbMC_CalcDynamicsByRampTime' );
	//LocalVars.State				:= MV_ERROR;
END_IF

// Call Fbs Cyclically
fbMC_CalcDynamicsByRampTime();
END_METHOD

METHOD MoveToStationByRampTime
VAR_INPUT
	DestinationStation	: REFERENCE TO Station;	
    Velocity     : LREAL;
    RampTime     : LREAL;
    Stiffness    : LREAL;
	Gap			 : LREAL;
END_VAR
VAR
	MotionParameters: MotionParameters_typ;
END_VAR
// This method internally calls MC_CalcDynamicsByRampTime from Tc2_MC2.lib
// https://infosys.beckhoff.com/content/1033/tcplclib_tc2_mc2/13611300875.html?id=1298283191705576852

fbMC_CalcDynamicsByRampTime(
	Velocity:= Velocity, 
	RampTime:= RampTime, 
	Stiffness:= Stiffness, 
	Error=> , 
	ErrorID=> , 
	Acceleration=> , 
	Deceleration=> , 
	Jerk=> );

MotionParameters.Velocity			:= Velocity;
MotionParameters.Acceleration		:= fbMC_CalcDynamicsByRampTime.Acceleration;
MotionParameters.Deceleration		:= fbMC_CalcDynamicsByRampTime.Deceleration;
MotionParameters.Jerk				:= fbMC_CalcDynamicsByRampTime.Jerk;
MotionParameters.Gap				:= Gap;
MotionParameters.Direction			:= Tc2_Mc2.MC_Direction.MC_Positive_Direction;

SUPER^.MotionParameters:= MotionParameters;
SUPER^.MoveToStation(DestinationStation);
END_METHOD

{attribute 'monitoring' := 'call'}
PROPERTY PositionLag : LREAL
GET
PositionLag:= _PositionLag;
END_GET
END_PROPERTY

END_FUNCTION_BLOCK

// ---- POUs/MAIN_LD.TcPOU
PROGRAM MAIN_LD
VAR	

	// ========= System Control / FSM Variables =========
	
	MainCommands 		: XTSCommands_typ; 		// command struct for cycling thru the state machine
	MainState    		: XTSStateMachine_enum;   	// enumeration for the Main state machine
	System				: Mediator;					// System-level control object

	// ========= Linked NC Variables & References =========
	
	Mover    			: ARRAY[1..GVL.NUM_MOVERS] OF Mover; 	// instantiation of Mover objects. Matches the number of movers on the system
	
	// ========= Objectives & Parameters =========

	ParameterSet		: MotionParameters_typ;
	
	MoverList			: ARRAY[0..GVL.NUM_MOVERLISTS-1] OF MoverList;
	PositionTrigger		: ARRAY[0..GVL.NUM_POSITIONTRIGGERS-1] OF PositionTrigger;
	Station				: ARRAY[0..GVL.NUM_STATIONS-1] OF Station;
	Track				: ARRAY[0..GVL.NUM_TRACKS] OF Track;
	Zone				: ARRAY[0..GVL.NUM_ZONES-1] OF Zone;
	
    // ========= Helper, State, & Index Variables =========
	
    i                	: UINT; 	// index variable; gets reused in various FOR loops
    n                	: UINT; 	// secondary index variable, for enabling movers
	
	// ========= Example Application Variables =========

    nextStation 			: USINT := 4;
                    	
    lowVelocity    			: LREAL := 200;  	// mm/s
    mediumVelocity 			: LREAL := 800;  	// mm/s
    highVelocity   			: LREAL := 1200; 	// mm/s
	
	StationTimer 			: ARRAY[0..GVL.NUM_STATIONS] OF TON; // timer blocks, for station dwells
	InitialParameterSet		: MotionParameters_typ;
	
	// ========= Additional Ladder Variables =========
	MS_Disabled						: BOOL;
	MS_Initializing					: BOOL;
	MS_Enabled						: BOOL;
	MS_Run							: BOOL;
	MS_Stopping						: BOOL;
	MS_Stopped						: BOOL;
	MS_Disabling					: BOOL;
	MS_Error						: BOOL;
	MS_Debug						: BOOL;
	
	MS_Enabled_StartReady			: BOOL;
	StationGroupInPosition			: BOOL;
	StationGroupMoversInPosition	: BOOL;
	Station1_TimerIn: BOOL;
END_VAR
VAR // added by the converter: edge detectors and wires of the graphical bodies
    _w1, _w2, _w3, _w4, _w5, _w6, _w7, _w8, _w9 : BOOL;
END_VAR

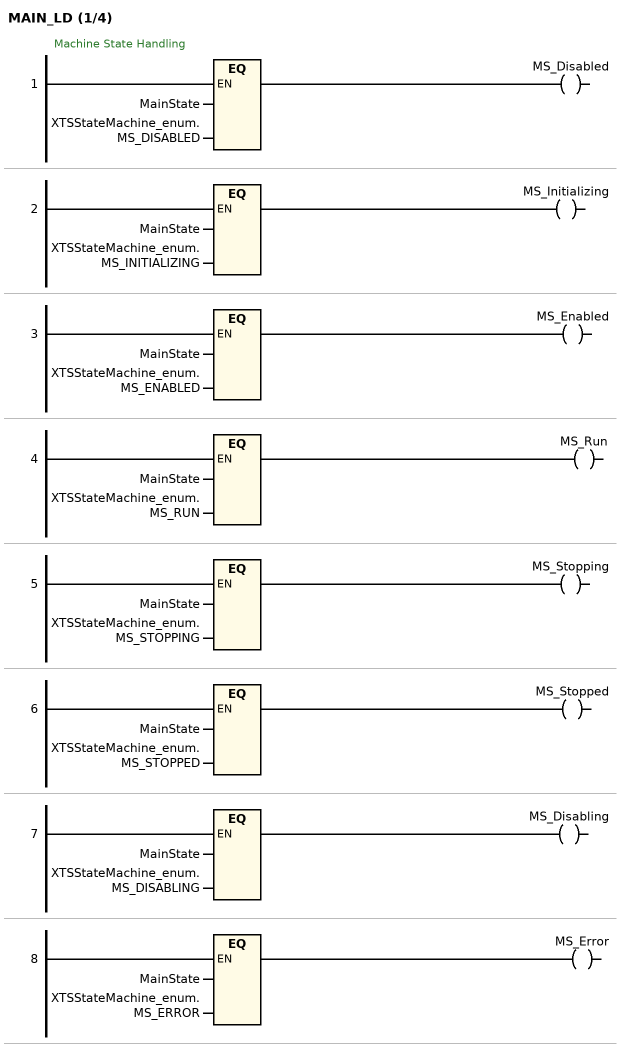
// NETWORK 1
// Machine State Handling
MS_Disabled := MainState = XTSStateMachine_enum.MS_DISABLED;

// NETWORK 2
MS_Initializing := MainState = XTSStateMachine_enum.MS_INITIALIZING;

// NETWORK 3
MS_Enabled := MainState = XTSStateMachine_enum.MS_ENABLED;

// NETWORK 4
MS_Run := MainState = XTSStateMachine_enum.MS_RUN;

// NETWORK 5
MS_Stopping := MainState = XTSStateMachine_enum.MS_STOPPING;

// NETWORK 6
MS_Stopped := MainState = XTSStateMachine_enum.MS_STOPPED;

// NETWORK 7
MS_Disabling := MainState = XTSStateMachine_enum.MS_DISABLING;

// NETWORK 8
MS_Error := MainState = XTSStateMachine_enum.MS_ERROR;

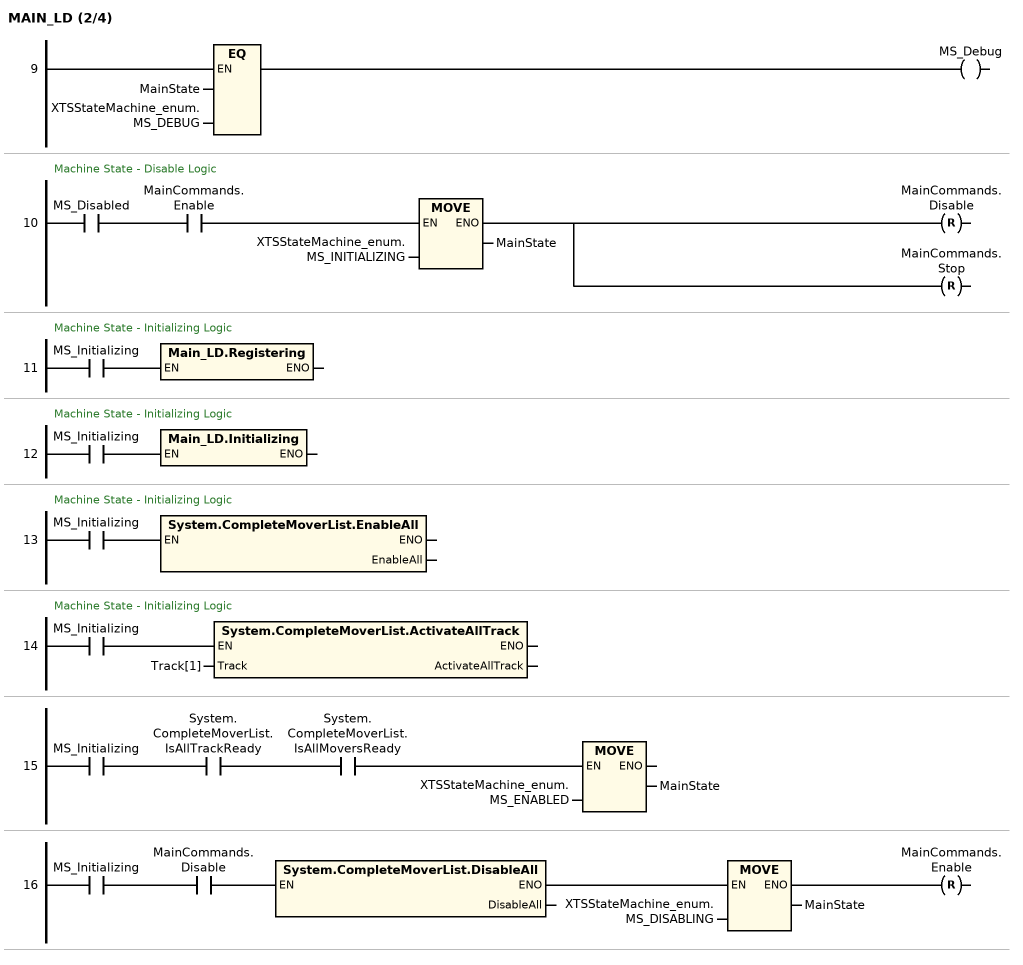
// NETWORK 9
MS_Debug := MainState = XTSStateMachine_enum.MS_DEBUG;

// NETWORK 10
// Machine State - Disable Logic
_w1 := MS_Disabled AND MainCommands.Enable;
IF _w1 THEN MainState := XTSStateMachine_enum.MS_INITIALIZING; END_IF
MainCommands.Disable R= _w1;
MainCommands.Stop R= _w1;

// NETWORK 11
// Machine State - Initializing Logic
IF MS_Initializing THEN Main_LD.Registering(); END_IF

// NETWORK 12
// Machine State - Initializing Logic
IF MS_Initializing THEN Main_LD.Initializing(); END_IF

// NETWORK 13
// Machine State - Initializing Logic
IF MS_Initializing THEN System.CompleteMoverList.EnableAll(); END_IF

// NETWORK 14
// Machine State - Initializing Logic
IF MS_Initializing THEN System.CompleteMoverList.ActivateAllTrack(Track := Track[1]); END_IF

// NETWORK 15
IF MS_Initializing AND System.CompleteMoverList.IsAllTrackReady AND System.CompleteMoverList.IsAllMoversReady THEN
    MainState := XTSStateMachine_enum.MS_ENABLED;
END_IF

// NETWORK 16
_w2 := MS_Initializing AND MainCommands.Disable;
IF _w2 THEN System.CompleteMoverList.DisableAll(); END_IF
IF _w2 THEN MainState := XTSStateMachine_enum.MS_DISABLING; END_IF
MainCommands.Enable R= _w2;

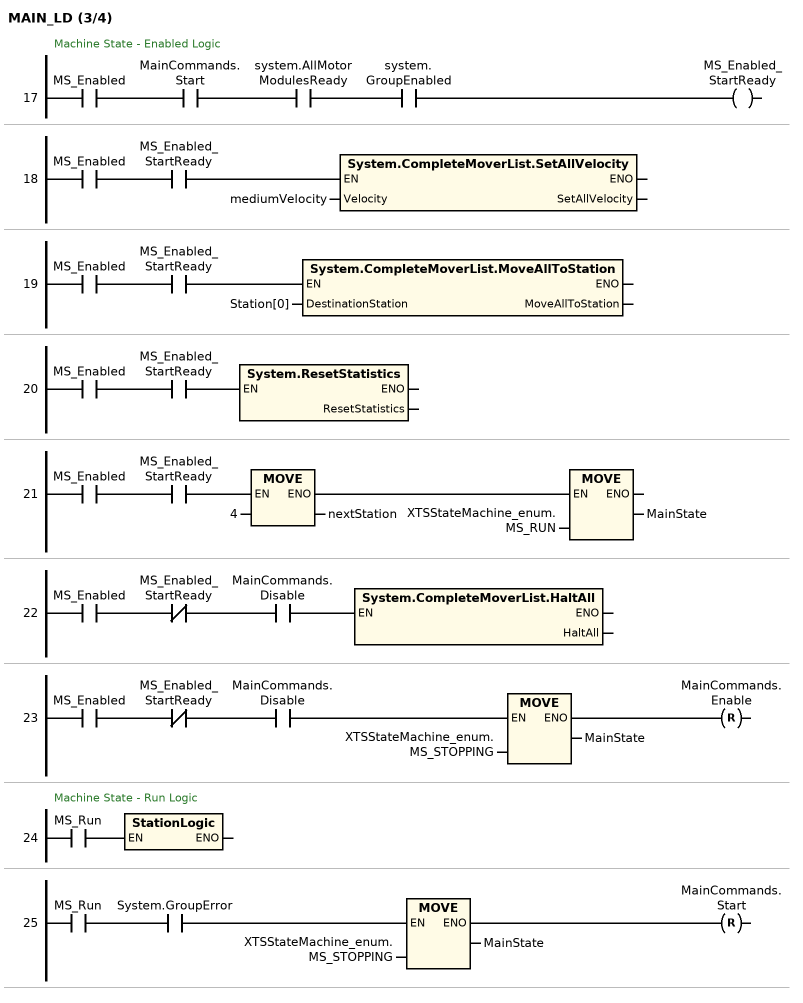
// NETWORK 17
// Machine State - Enabled Logic
MS_Enabled_StartReady := MS_Enabled AND MainCommands.Start AND system.AllMotorModulesReady AND system.GroupEnabled;

// NETWORK 18
IF MS_Enabled AND MS_Enabled_StartReady THEN
    System.CompleteMoverList.SetAllVelocity(Velocity := mediumVelocity);
END_IF

// NETWORK 19
IF MS_Enabled AND MS_Enabled_StartReady THEN
    System.CompleteMoverList.MoveAllToStation(DestinationStation := Station[0]);
END_IF

// NETWORK 20
IF MS_Enabled AND MS_Enabled_StartReady THEN System.ResetStatistics(); END_IF

// NETWORK 21
_w3 := MS_Enabled AND MS_Enabled_StartReady;
IF _w3 THEN nextStation := 4; END_IF
IF _w3 THEN MainState := XTSStateMachine_enum.MS_RUN; END_IF

// NETWORK 22
IF MS_Enabled AND NOT MS_Enabled_StartReady AND MainCommands.Disable THEN
    System.CompleteMoverList.HaltAll();
END_IF

// NETWORK 23
_w4 := MS_Enabled AND NOT MS_Enabled_StartReady AND MainCommands.Disable;
IF _w4 THEN MainState := XTSStateMachine_enum.MS_STOPPING; END_IF
MainCommands.Enable R= _w4;

// NETWORK 24
// Machine State - Run Logic
IF MS_Run THEN StationLogic(); END_IF

// NETWORK 25
_w5 := MS_Run AND System.GroupError;
IF _w5 THEN MainState := XTSStateMachine_enum.MS_STOPPING; END_IF
MainCommands.Start R= _w5;

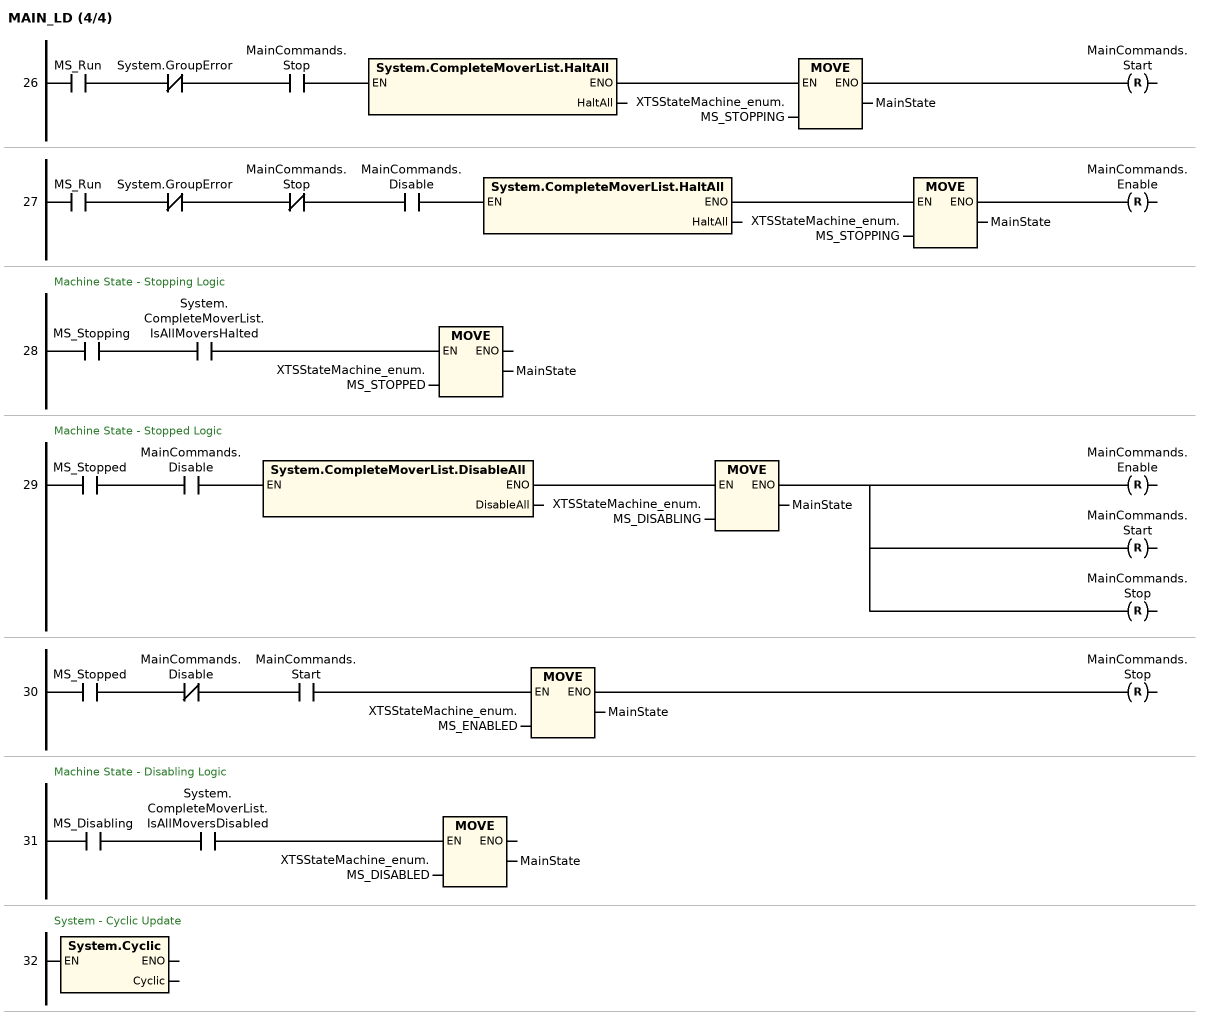
// NETWORK 26
_w6 := MS_Run AND NOT System.GroupError AND MainCommands.Stop;
IF _w6 THEN System.CompleteMoverList.HaltAll(); END_IF
IF _w6 THEN MainState := XTSStateMachine_enum.MS_STOPPING; END_IF
MainCommands.Start R= _w6;

// NETWORK 27
_w7 := MS_Run AND NOT System.GroupError AND NOT MainCommands.Stop AND MainCommands.Disable;
IF _w7 THEN System.CompleteMoverList.HaltAll(); END_IF
IF _w7 THEN MainState := XTSStateMachine_enum.MS_STOPPING; END_IF
MainCommands.Enable R= _w7;

// NETWORK 28
// Machine State - Stopping Logic
IF MS_Stopping AND System.CompleteMoverList.IsAllMoversHalted THEN
    MainState := XTSStateMachine_enum.MS_STOPPED;
END_IF

// NETWORK 29
// Machine State - Stopped Logic
_w8 := MS_Stopped AND MainCommands.Disable;
IF _w8 THEN System.CompleteMoverList.DisableAll(); END_IF
IF _w8 THEN MainState := XTSStateMachine_enum.MS_DISABLING; END_IF
MainCommands.Enable R= _w8;
MainCommands.Start R= _w8;
MainCommands.Stop R= _w8;

// NETWORK 30
_w9 := MS_Stopped AND NOT MainCommands.Disable AND MainCommands.Start;
IF _w9 THEN MainState := XTSStateMachine_enum.MS_ENABLED; END_IF
MainCommands.Stop R= _w9;

// NETWORK 31
// Machine State - Disabling Logic
IF MS_Disabling AND System.CompleteMoverList.IsAllMoversDisabled THEN
    MainState := XTSStateMachine_enum.MS_DISABLED;
END_IF

// NETWORK 32
// System - Cyclic Update
System.Cyclic();

ACTION Initializing:


	// Initialize station positions
	Station[0].Position 		:= 5;
	Station[1].Position 		:= 750;
	Station[2].Position 		:= 1200;
	Station[3].Position 		:= 1300;
	Station[4].Position 		:= 1400;

	PositionTrigger[0].Position := 1500;
	PositionTrigger[1].Position := 2000;
	PositionTrigger[2].Position := 3500;

	Zone[0].StartPosition		:= 3750;
	Zone[0].EndPosition   		:= 750;

	Zone[1].StartPosition 		:= 750;
	Zone[1].EndPosition   		:= 1750;

	Zone[2].StartPosition 		:= 1750;
	Zone[2].EndPosition   		:= 2750;

	Zone[3].StartPosition		:= 2750;
	Zone[3].EndPosition   		:= 3750;

	InitialParameterSet.Velocity		:= 1000;		// mm/s
	InitialParameterSet.Acceleration	:= 10_000;		// mm/s2
	InitialParameterSet.Deceleration	:= 10_000;		// mm/s2
	InitialParameterSet.Jerk			:= 100_000;		// mm/s3
	InitialParameterSet.Gap				:= 85;			// mm
	InitialParameterSet.Direction		:= mcDirectionPositive;	
	
	System.CompleteMoverList.ApplyAllParameterSet( InitialParameterSet );
END_ACTION

ACTION Registering:
	

		// Add all Movers to the Mediator
		FOR i := 1 TO GVL.NUM_MOVERS DO
			System.AddMover( Mover[i] );
		END_FOR
	
		// Add all Mover Lists to the Mediator
		FOR i := 0 TO GVL.NUM_MOVERLISTS - 1 DO
			System.AddMoverList( MoverList[i] );
		END_FOR
		
		// Add all PositionTriggers to the Mediator
		FOR i := 0 TO GVL.NUM_POSITIONTRIGGERS - 1 DO
			System.AddPositionTrigger( PositionTrigger[i] );
		END_FOR
		
		// Add all Stations to the Mediator
		FOR i := 0 TO GVL.NUM_STATIONS - 1 DO
			System.AddStation( Station[i] );
		END_FOR
		
		// Add all Tracks to the Mediator
		// note track zero is a special case, so the loop is one larger than the rest of the initalization loops
		FOR i := 0 TO GVL.NUM_TRACKS DO
			Track[i].Id := UINT_TO_INT(i);
			System.AddTrack( Track[i] );
		END_FOR
		
		// Add all Zones to the Mediator
		FOR i := 0 TO GVL.NUM_ZONES - 1 DO
			System.AddZone( Zone[i] );
		END_FOR
END_ACTION

ACTION StationLogic:
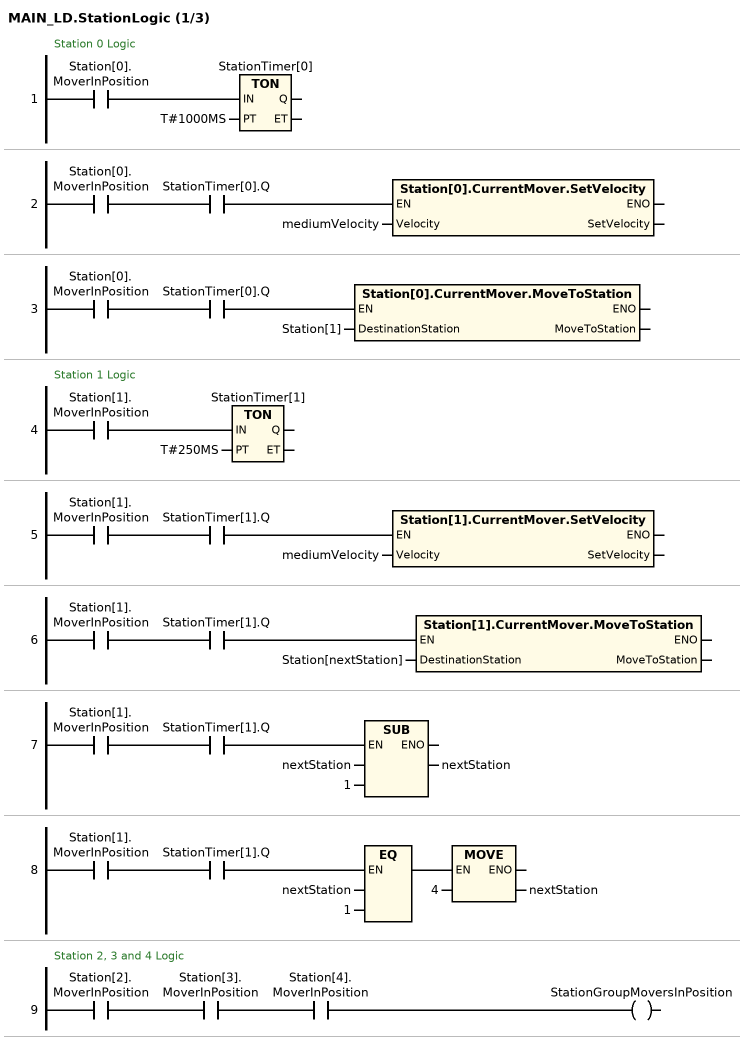
// NETWORK 1
// Station 0 Logic
StationTimer[0](IN := Station[0].MoverInPosition, PT := T#1000MS); // TON

// NETWORK 2
IF Station[0].MoverInPosition AND StationTimer[0].Q THEN
    Station[0].CurrentMover.SetVelocity(Velocity := mediumVelocity);
END_IF

// NETWORK 3
IF Station[0].MoverInPosition AND StationTimer[0].Q THEN
    Station[0].CurrentMover.MoveToStation(DestinationStation := Station[1]);
END_IF

// NETWORK 4
// Station 1 Logic
StationTimer[1](IN := Station[1].MoverInPosition, PT := T#250MS); // TON

// NETWORK 5
IF Station[1].MoverInPosition AND StationTimer[1].Q THEN
    Station[1].CurrentMover.SetVelocity(Velocity := mediumVelocity);
END_IF

// NETWORK 6
IF Station[1].MoverInPosition AND StationTimer[1].Q THEN
    Station[1].CurrentMover.MoveToStation(DestinationStation := Station[nextStation]);
END_IF

// NETWORK 7
IF Station[1].MoverInPosition AND StationTimer[1].Q THEN nextStation := nextStation - 1; END_IF

// NETWORK 8
IF Station[1].MoverInPosition AND StationTimer[1].Q AND nextStation = 1 THEN nextStation := 4; END_IF

// NETWORK 9
// Station 2, 3 and 4 Logic
StationGroupMoversInPosition := Station[2].MoverInPosition AND Station[3].MoverInPosition AND Station[4].MoverInPosition;

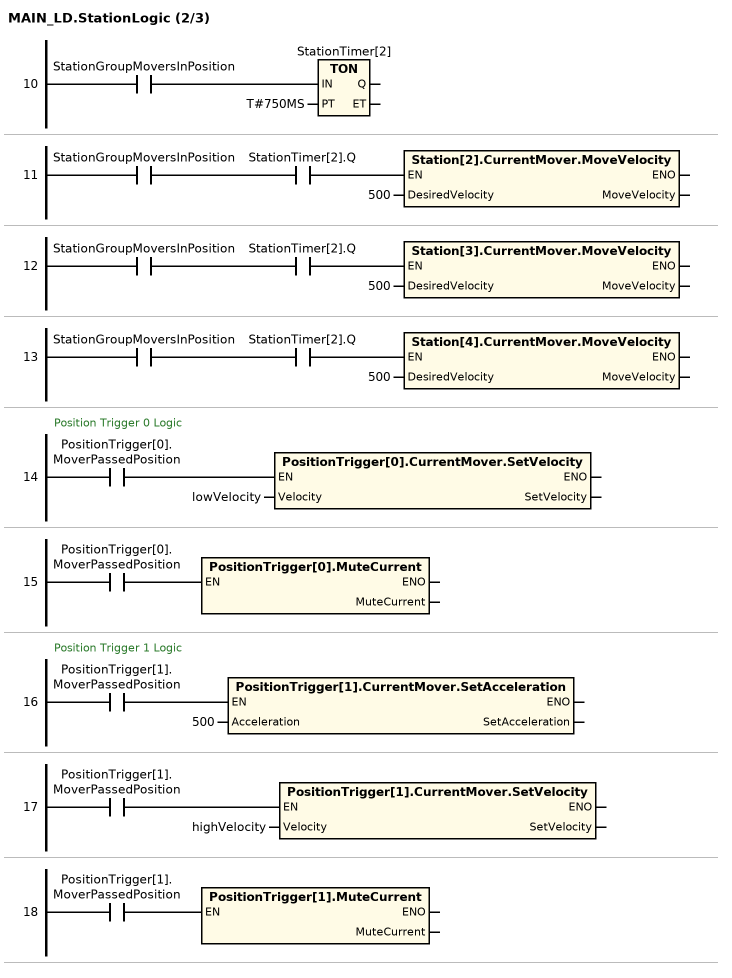
// NETWORK 10
StationTimer[2](IN := StationGroupMoversInPosition, PT := T#750MS); // TON

// NETWORK 11
IF StationGroupMoversInPosition AND StationTimer[2].Q THEN
    Station[2].CurrentMover.MoveVelocity(DesiredVelocity := 500);
END_IF

// NETWORK 12
IF StationGroupMoversInPosition AND StationTimer[2].Q THEN
    Station[3].CurrentMover.MoveVelocity(DesiredVelocity := 500);
END_IF

// NETWORK 13
IF StationGroupMoversInPosition AND StationTimer[2].Q THEN
    Station[4].CurrentMover.MoveVelocity(DesiredVelocity := 500);
END_IF

// NETWORK 14
// Position Trigger 0 Logic
IF PositionTrigger[0].MoverPassedPosition THEN
    PositionTrigger[0].CurrentMover.SetVelocity(Velocity := lowVelocity);
END_IF

// NETWORK 15
IF PositionTrigger[0].MoverPassedPosition THEN PositionTrigger[0].MuteCurrent(); END_IF

// NETWORK 16
// Position Trigger 1 Logic
IF PositionTrigger[1].MoverPassedPosition THEN
    PositionTrigger[1].CurrentMover.SetAcceleration(Acceleration := 500);
END_IF

// NETWORK 17
IF PositionTrigger[1].MoverPassedPosition THEN
    PositionTrigger[1].CurrentMover.SetVelocity(Velocity := highVelocity);
END_IF

// NETWORK 18
IF PositionTrigger[1].MoverPassedPosition THEN PositionTrigger[1].MuteCurrent(); END_IF

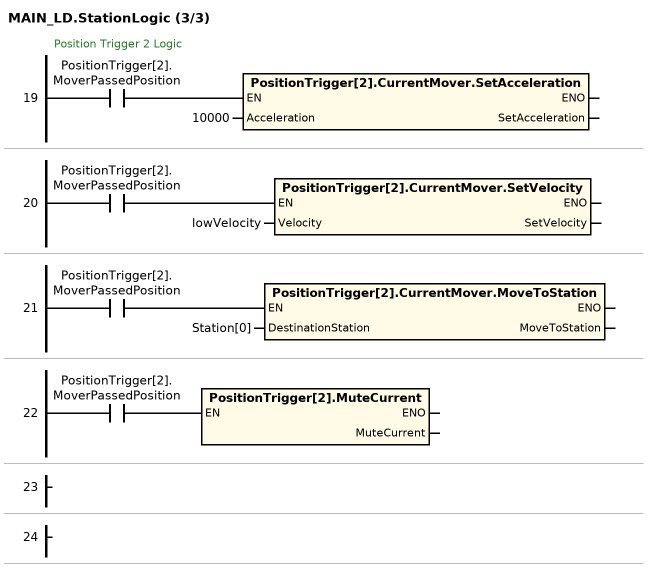
// NETWORK 19
// Position Trigger 2 Logic
IF PositionTrigger[2].MoverPassedPosition THEN
    PositionTrigger[2].CurrentMover.SetAcceleration(Acceleration := 10000);
END_IF

// NETWORK 20
IF PositionTrigger[2].MoverPassedPosition THEN
    PositionTrigger[2].CurrentMover.SetVelocity(Velocity := lowVelocity);
END_IF

// NETWORK 21
IF PositionTrigger[2].MoverPassedPosition THEN
    PositionTrigger[2].CurrentMover.MoveToStation(DestinationStation := Station[0]);
END_IF

// NETWORK 22
IF PositionTrigger[2].MoverPassedPosition THEN PositionTrigger[2].MuteCurrent(); END_IF

// NETWORK 23

// NETWORK 24
END_ACTION

END_PROGRAM

// ---- GlobalTextList.TcGTLO
TEXTLIST GlobalTextList
  453 = '%4.0f mm/s'
  517 = 'Disable'
  232 = 'Enable'
  434 = 'High Velocity'
  919 = 'Low Velocity'
  500 = 'Medium Velocity'
  393 = 'Start'
  920 = 'Stop'
END_TEXTLIST

// ---- VISUs/Controls.TcVIS
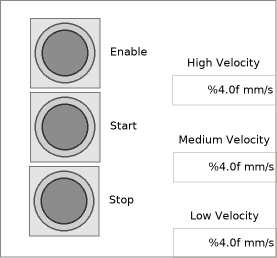
VISUALIZATION Controls  // 277x258
    PushSwitchLed (30,18 70x70), variable: MAIN.MainCommands.Enable, behaviour: TOGGLE, style: Switch-PushSwitchLed-Gray
    Label (107,37 75x30), "Enable"
    Label (107,111 75x30), "Start"
    PushSwitchLed (30,92 70x70), variable: MAIN.MainCommands.Start, behaviour: TOGGLE, style: Switch-PushSwitchLed-Gray
    Label (106,185 75x30), "Stop"
    PushSwitchLed (29,166 70x70), variable: MAIN.MainCommands.Stop, behaviour: TOGGLE, style: Switch-PushSwitchLed-Gray
    Textfield (172,75 104x30), "%4.0f mm/s", text variable: MAIN.highVelocity
        OnMouseClick: write the text variable via VisuDialogs.Numpad, min 1, max 2000, format %f.0
    Label (175,54 97x18), "High Velocity"
    Textfield (173,152 104x30), "%4.0f mm/s", text variable: MAIN.mediumVelocity
        OnMouseClick: write the text variable via VisuDialogs.Numpad, min 1, max 2000, format %f.0
    Label (176,131 97x18), "Medium Velocity"
    Textfield (173,228 104x30), "%4.0f mm/s", text variable: MAIN.lowVelocity
        OnMouseClick: write the text variable via VisuDialogs.Numpad, min 1, max 2000, format %f.0
    Label (176,207 97x18), "Low Velocity"
END_VISUALIZATION

// ---- VISUs/DiagnosticVisu.TcVIS
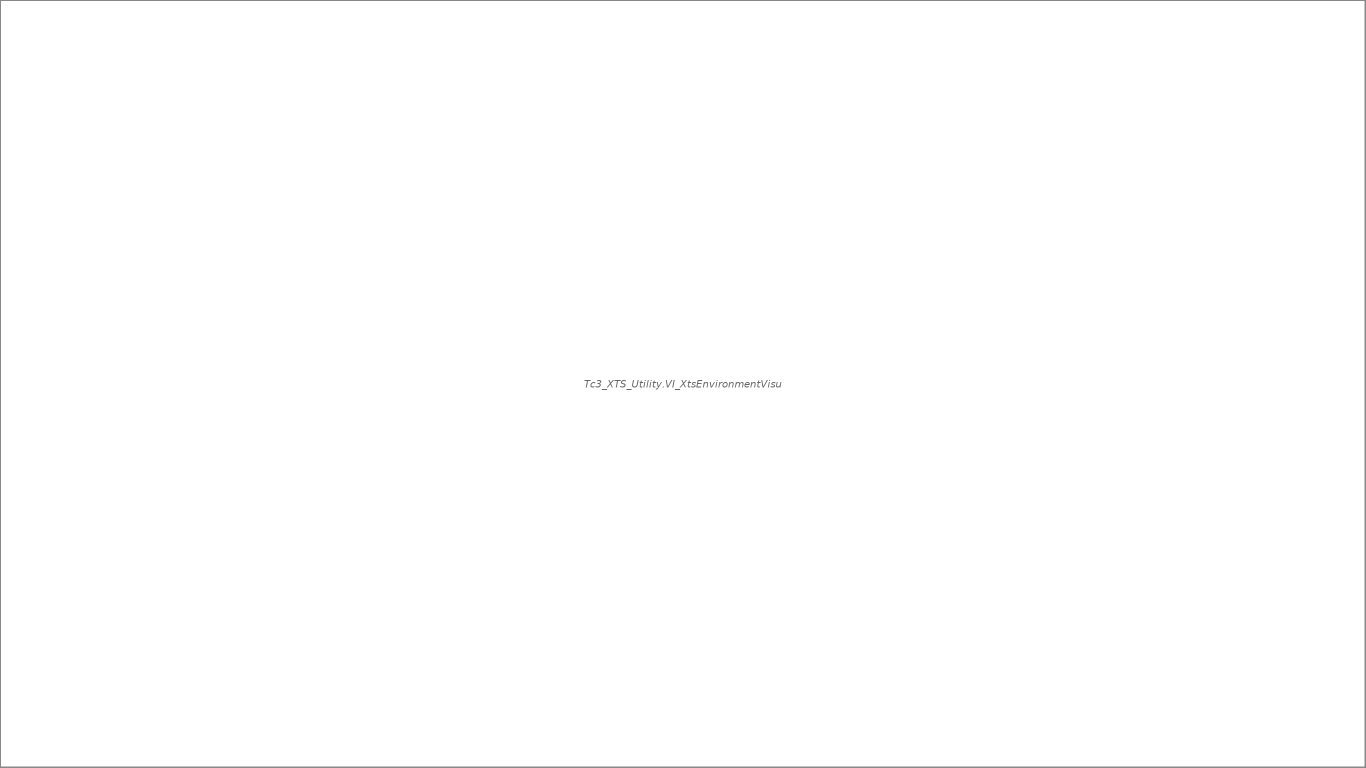
VISUALIZATION DiagnosticVisu  // 1366x768
    Frame (0,0 1366x768)
        shows Tc3_XTS_Utility.VI_XtsEnvironmentVisu()
END_VISUALIZATION
